TYPE ST_MachineState :
STRUCT

	bStartup	 : BOOL;		
	bStartupDone : BOOL;
	bAborting 	 : BOOL;
	bResetting	 : BOOL;
	bStarting	 : BOOL;
	bRunning	 : BOOL;

END_STRUCT
END_TYPE

(* stored: Version 1.1.0.1, ProductVersion 3.1.4024.4
   DUT ST_MachineState: Id {24ec17bb-f366-4b25-b13e-a294e7e9931d} *)
